// TwinCAT 3 PLC project PLC
// ProgramVersion: 3.1.4026.21
// libraries:
//   Tc2_Standard, * (Beckhoff Automation GmbH)
//   Tc2_System, * (Beckhoff Automation GmbH)
//   Tc2_Utilities, * (Beckhoff Automation GmbH)
// project tree:
//   / PlcTask.TcTTO
//   POUs/ Echange_OPCUA.TcPOU, MAIN.TcPOU

CONFIGURATION PLC
    RESOURCE PLC ON TwinCAT3
        TASK PlcTask(INTERVAL := T#10ms, PRIORITY := 20);
        PROGRAM MAIN WITH PlcTask : MAIN;
    END_RESOURCE
END_CONFIGURATION

// ---- POUs/MAIN.TcPOU
PROGRAM MAIN
VAR
END_VAR

Echange_OPCUA();

END_PROGRAM

// ---- POUs/Echange_OPCUA.TcPOU
PROGRAM Echange_OPCUA
VAR
	Ton_NT_GetTime:Ton;
	fbGetTime:NT_GetTime;
	
	{attribute 'OPC.UA.DA' := '1'}
	stTIMESTR: Tc2_Utilities.TIMESTRUCT;
END_VAR

fbGetTime(
	NETID:= '', 
	START:= Ton_NT_GetTime.Q, 
	TMOUT:= DEFAULT_ADS_TIMEOUT, 
	BUSY=> , 
	ERR=> , 
	ERRID=> , 
	TIMESTR=> stTIMESTR);
	
	
Ton_NT_GetTime(IN:= NOT fbGetTime.BUSY , PT:=T#500MS , Q=> , ET=> );

END_PROGRAM
